(* PLC project CoDeSys External Library Template, WAGO e!COCKPIT e!COCKPIT, author 3S - Smart Software Solutions GmbH *)
(* stored: creationDateTime 2019-10-29T12:22:40.8911777, version 3.5.5.30, modificationDateTime 2019-10-24T14:40:07.960949, organization 3S - Smart Software Solutions GmbH *)
(* Library project template with all possible element types, docu and a sample project structure *)

(* funkcja do kompleksowej obróbki komunikatu *)
FUNCTION fnKomunikatInOut : BOOL
  VAR_INPUT
    xStringNaStrukture : BOOL;  (* rozkaz rozbicia pełnego komunikatu na cząstki *)
    xStringUpdateZeStruktury : BOOL;
    xStrukturyNaString : BOOL;
    xWyczyscStrukture : BOOL;
    xAktualizujZnacznikCzasu : BOOL;  (* rozkaz zaktualizowania znacznika czasu - działa we wszystkich konfiguracjach *)
    xAktualizujDlugoscDanych : BOOL;
  END_VAR
  VAR_IN_OUT
    sKomunikat : alSTRINGKomunikat;
    typKomunikat : typKomunikat;
    intBlad : INT;
  END_VAR
  VAR
    sKomunikatTemp : alSTRINGKomunikat;
  END_VAR

            IF xWyczyscStrukture AND xStringNaStrukture THEN
	fnKomunikatInOutZeruj(typKomunikat);
END_IF
IF xStrukturyNaString THEN
	sKomunikat := CONCAT(typKomunikat.sZnacznik , typKomunikat.sTypKomunikatu);
	sKomunikat := CONCAT(sKomunikat , typKomunikat.sMnemonikWlasciciela);
	sKomunikat := CONCAT(sKomunikat , typKomunikat.sMnemonikWlascicielaExt);
	sKomunikat := CONCAT(sKomunikat , typKomunikat.sMACAdres);	
	IF typKomunikat.sIDZrodla = '' THEN
		sKomunikat := CONCAT(sKomunikat , typKomunikat.sIDZrodlaLokalizacja);
		sKomunikat := CONCAT(sKomunikat , typKomunikat.sIDZrodlaUrzadzenie);
		typKomunikat.sIDZrodla := CONCAT(typKomunikat.sIDZrodlaLokalizacja , typKomunikat.sIDZrodlaUrzadzenie);
		ELSE
		sKomunikat := CONCAT(sKomunikat , typKomunikat.sIDZrodla);
	END_IF
	IF typKomunikat.sIDPrzeznaczenia = '' THEN	
		sKomunikat := CONCAT(sKomunikat , typKomunikat.sIDPrzeznaczeniaLokalizacja);
		sKomunikat := CONCAT(sKomunikat , typKomunikat.sIDPrzeznaczeniaUrzadzenie);
		typKomunikat.sIDPrzeznaczenia := CONCAT(typKomunikat.sIDPrzeznaczeniaLokalizacja , typKomunikat.sIDPrzeznaczeniaUrzadzenie);
		ELSE
		sKomunikat := CONCAT(sKomunikat , typKomunikat.sIDPrzeznaczenia);		
	END_IF
	IF typKomunikat.sDlugoscPolaDanych = '' OR xAktualizujDlugoscDanych THEN
		sKomunikat := CONCAT(sKomunikat ,  fnKonwersjaINT_STRING(intWartosc := LEN(typKomunikat.sDane) , intIloscZnakow := 3));
		typKomunikat.sDlugoscPolaDanych := fnKonwersjaINT_STRING(intWartosc := LEN(typKomunikat.sDane) , intIloscZnakow := 3);
		ELSE
		sKomunikat := CONCAT(sKomunikat , typKomunikat.sDlugoscPolaDanych);
	END_IF
	IF typKomunikat.sMarkerCzasowy = '' OR xAktualizujZnacznikCzasu THEN
		sKomunikat := CONCAT(sKomunikat , fnCzasUTC());
		typKomunikat.sMarkerCzasowy := fnCzasUTC();
		ELSE		
		sKomunikat := CONCAT(sKomunikat , typKomunikat.sMarkerCzasowy);
	END_IF
	sKomunikat := CONCAT(sKomunikat , typKomunikat.sRezerwa);
	sKomunikat := CONCAT(sKomunikat , typKomunikat.sDane);
END_IF

IF xStringNaStrukture OR xStringUpdateZeStruktury THEN
	IF typKomunikat.sZnacznik <> '' AND xStringUpdateZeStruktury THEN
		sKomunikat := CONCAT(typKomunikat.sZnacznik , MID(sKomunikat , LEN(sKomunikat) - 1 , 2));
		ELSE
		typKomunikat.sZnacznik := LEFT(sKomunikat , 1);
	END_IF
	IF typKomunikat.sTypKomunikatu <> '' AND xStringUpdateZeStruktury THEN
		sKomunikatTemp := LEFT(sKomunikat , 1);
		sKomunikat := CONCAT(typKomunikat.sTypKomunikatu , MID(sKomunikat , LEN(sKomunikat) - 2 , 3));
		sKomunikat := CONCAT(sKomunikatTemp , sKomunikat);
		ELSE
		typKomunikat.sTypKomunikatu := MID(SKomunikat , 1 , 2);
	END_IF
	IF typKomunikat.sMnemonikWlasciciela <> '' AND xStringUpdateZeStruktury THEN
		sKomunikatTemp := LEFT(sKomunikat , 2);
		sKomunikat := CONCAT(typKomunikat.sMnemonikWlasciciela , MID(sKomunikat , LEN(sKomunikat) - 5 , 6));
		sKomunikat := CONCAT(sKomunikatTemp , sKomunikat);
		ELSE
		typKomunikat.sMnemonikWlasciciela := MID(sKomunikat , 3 , 3);
	END_IF
	IF typKomunikat.sMnemonikWlascicielaExt <> '' AND xStringUpdateZeStruktury THEN
		sKomunikatTemp := LEFT(sKomunikat , 5);
		sKomunikat := CONCAT(typKomunikat.sMnemonikWlascicielaExt , MID(sKomunikat , LEN(sKomunikat) - 6 , 7));
		sKomunikat := CONCAT(sKomunikatTemp , sKomunikat);
		ELSE
		typKomunikat.sMnemonikWlascicielaExt := MID(Skomunikat , 1 , 6);
	END_IF
	IF typKomunikat.sMACAdres <> '' AND xStringUpdateZeStruktury THEN
		sKomunikatTemp := LEFT(sKomunikat , 6);
		sKomunikat := CONCAT(typKomunikat.sMnemonikWlascicielaExt , MID(sKomunikat , LEN(sKomunikat) - 12 , 13));
		sKomunikat := CONCAT(sKomunikatTemp , sKomunikat);
		ELSE
		typKomunikat.sMACAdres := MID(sKomunikat , 6 , 7);
	END_IF
	IF typKomunikat.sIDZrodla <> '' AND xStringUpdateZeStruktury THEN
		sKomunikatTemp := LEFT(sKomunikat , 12);
		sKomunikat := CONCAT(typKomunikat.sIDZrodla , MID(sKomunikat , LEN(sKomunikat) - 28 , 29));
		sKomunikat := CONCAT(sKomunikatTemp , sKomunikat);
		ELSE
		typKomunikat.sIDZrodla := MID(sKomunikat , 16 , 13);
	END_IF
	IF typKomunikat.sIDZrodlaLokalizacja <> '' AND xStringUpdateZeStruktury THEN
		sKomunikatTemp := LEFT(sKomunikat , 12);
		sKomunikat := CONCAT(typKomunikat.sIDZrodlaLokalizacja , MID(sKomunikat , LEN(sKomunikat) - 24 , 25));
		sKomunikat := CONCAT(sKomunikatTemp , sKomunikat);
		ELSE
		typKomunikat.sIDZrodlaLokalizacja := MID(SKomunikat , 12 , 13);
	END_IF
	IF typKomunikat.sIDZrodlaUrzadzenie <> '' AND xStringUpdateZeStruktury THEN
		sKomunikatTemp := LEFT(sKomunikat , 24);
		sKomunikat := CONCAT(typKomunikat.sIDZrodlaUrzadzenie , MID(sKomunikat , LEN(sKomunikat) - 28 , 29));
		sKomunikat := CONCAT(sKomunikatTemp , sKomunikat);
		ELSE
		typKomunikat.sIDZrodlaUrzadzenie := MID(SKomunikat , 4 , 25);		
	END_IF
	IF typKomunikat.sIDPrzeznaczenia <> '' AND xStringUpdateZeStruktury THEN
		sKomunikatTemp := LEFT(sKomunikat , 28);
		sKomunikat := CONCAT(typKomunikat.sIDPrzeznaczenia , MID(sKomunikat , LEN(sKomunikat) - 44 ,45));
		sKomunikat := CONCAT(sKomunikatTemp , sKomunikat);
		ELSE
		typKomunikat.sIDPrzeznaczenia := MID(SKomunikat , 16 , 29);
	END_IF
	IF typKomunikat.sIDPrzeznaczeniaLokalizacja <> '' AND xStringUpdateZeStruktury THEN
		sKomunikatTemp := LEFT(sKomunikat , 28);
		sKomunikat := CONCAT(typKomunikat.sIDPrzeznaczeniaLokalizacja , MID(sKomunikat , LEN(sKomunikat) - 40 ,41));
		sKomunikat := CONCAT(sKomunikatTemp , sKomunikat);
		ELSE
		typKomunikat.sIDPrzeznaczeniaLokalizacja := MID(SKomunikat , 12 , 29);
	END_IF
	IF typKomunikat.sIDPrzeznaczeniaUrzadzenie <> '' AND xStringUpdateZeStruktury THEN
		sKomunikatTemp := LEFT(sKomunikat , 40);
		sKomunikat := CONCAT(typKomunikat.sIDPrzeznaczeniaUrzadzenie , MID(sKomunikat , LEN(sKomunikat) - 44 ,45));
		sKomunikat := CONCAT(sKomunikatTemp , sKomunikat);
		ELSE
		typKomunikat.sIDPrzeznaczeniaUrzadzenie := MID(SKomunikat , 4 , 41);
	END_IF
	IF typKomunikat.sMarkerCzasowy <> '' AND xStringUpdateZeStruktury THEN
		IF xAktualizujZnacznikCzasu THEN
			sKomunikatTemp := LEFT(sKomunikat , 47);
			sKomunikat := CONCAT(fnCzasUTC() , MID(sKomunikat , LEN(sKomunikat) - 76 , 77));			
			sKomunikat := CONCAT(sKomunikatTemp , sKomunikat);
			ELSE
			sKomunikatTemp := LEFT(sKomunikat , 47);
			sKomunikat := CONCAT(typKomunikat.sMarkerCzasowy , MID(sKomunikat , LEN(sKomunikat) - 76 , 77));
			sKomunikat := CONCAT(sKomunikatTemp , sKomunikat);
		END_IF
		ELSE
		typKomunikat.sMarkerCzasowy := MID(SKomunikat , 29 , 48);
	END_IF
	IF typKomunikat.sRezerwa <> '' AND xStringUpdateZeStruktury THEN
		sKomunikatTemp := LEFT(sKomunikat , 76);
		sKomunikat := CONCAT(typKomunikat.sRezerwa , MID(sKomunikat , LEN(sKomunikat) - 82 , 83));
		sKomunikat := CONCAT(sKomunikatTemp , sKomunikat);
		ELSE
		typKomunikat.sRezerwa := MID(SKomunikat , 6 , 77);
	END_IF
	IF typKomunikat.sDane <> '' AND xStringUpdateZeStruktury THEN
		sKomunikatTemp := LEFT(sKomunikat , 82);
		sKomunikat := CONCAT(sKomunikatTemp , typKomunikat.sDane);
		ELSE
		typKomunikat.sDane := RIGHT(sKomunikat ,  LEN(sKomunikat) - 82);
	END_IF
	IF typKomunikat.sDlugoscPolaDanych <> '' AND xStringUpdateZeStruktury THEN
		IF xAktualizujDlugoscDanych THEN
			sKomunikatTemp := LEFT(sKomunikat , 44);
			sKomunikat := CONCAT(fnKonwersjaINT_STRING(intWartosc := LEN(typKomunikat.sDane) , intIloscZnakow := 3) , MID(sKomunikat , LEN(sKomunikat) - 47 , 48));
			sKomunikat := CONCAT(sKomunikatTemp , sKomunikat);
		ELSE
			sKomunikatTemp := LEFT(sKomunikat , 44);
			sKomunikat := CONCAT(typKomunikat.sDlugoscPolaDanych , MID(sKomunikat , LEN(sKomunikat) - 47 , 48));
			sKomunikat := CONCAT(sKomunikatTemp , sKomunikat);
		END_IF
		ELSE
		typKomunikat.sDlugoscPolaDanych := MID(SKomunikat , 3 , 45);
	END_IF
END_IF

          
END_FUNCTION
